(* IEC 61131-3 sources: BombaAutomatica/BOMBA_CASA/build, 2 files *)

(* ---- plc.st ---- *)
TYPE
  LOGLEVEL : (CRITICAL, WARNING, INFO, DEBUG) := INFO;
END_TYPE

FUNCTION_BLOCK LOGGER
  VAR_INPUT
    TRIG : BOOL;
    MSG : STRING;
    LEVEL : LOGLEVEL := INFO;
  END_VAR
  VAR
    TRIG0 : BOOL;
  END_VAR

  IF TRIG AND NOT TRIG0 THEN
  {{
   LogMessage(GetFbVar(LEVEL),(char*)GetFbVar(MSG, .body),GetFbVar(MSG, .len));
  }}
  END_IF;
  TRIG0:=TRIG;
END_FUNCTION_BLOCK

PROGRAM Auto_bombas
  VAR
    Bomba_calle : BOOL;
    Flotador_cisterna : BOOL;
    Sensor_presion : BOOL;
    Arranque_bomba_calle : BOOL;
    Arranque_bomba_tinaco : BOOL;
    Sensor_tinaco : BOOL;
    Sensor_flujo : BOOL;
    TON0 : TON;
    TON1 : TIME := T#5s;
  END_VAR

  TON0(IN := NOT(Sensor_presion) AND Sensor_flujo AND NOT(Flotador_cisterna) AND Arranque_bomba_calle, PT := TON1);
  Bomba_calle := TON0.Q;
END_PROGRAM

CONFIGURATION Config0

  RESOURCE Res0 ON PLC
    TASK task0(INTERVAL := T#20ms,PRIORITY := 0);
    PROGRAM instance0 WITH task0 : Auto_bombas;
  END_RESOURCE
END_CONFIGURATION

(* ---- generated_plc.st ---- *)
PROGRAM Auto_bombas
  VAR
    Bomba_calle : BOOL;
    Flotador_cisterna : BOOL;
    Sensor_presion : BOOL;
    Arranque_bomba_calle : BOOL;
    Arranque_bomba_tinaco : BOOL;
    Sensor_tinaco : BOOL;
    Sensor_flujo : BOOL;
    TON0 : TON;
    TON1 : TIME := T#5s;
  END_VAR

  TON0(IN := NOT(Sensor_presion) AND Sensor_flujo AND NOT(Flotador_cisterna) AND Arranque_bomba_calle, PT := TON1);
  Bomba_calle := TON0.Q;
END_PROGRAM

CONFIGURATION Config0

  RESOURCE Res0 ON PLC
    TASK task0(INTERVAL := T#20ms,PRIORITY := 0);
    PROGRAM instance0 WITH task0 : Auto_bombas;
  END_RESOURCE
END_CONFIGURATION
